PROGRAM Stn054_29_EmptyPuckStorageMergeGrn
VAR
	{attribute 'TcLinkToOSO' := '	
			.iBufferFull :=  <0,1,3>TIIB[N56S00 (AL1332)]^N56S05 (AL2341)^TxPDO^input byte 2'}
	fbConvMerge: FB_ConvMerge_RemoteOutput;
	
	{attribute 'TcLinkToOSO' := '
			<0,1,3>TIIB[N56S00 (AL1332)]^N56S05 (AL2341)^TxPDO^input byte 2'}
	iBufferFull AT %I*: BOOL;

END_VAR

//  This code instantiates a component that is implimented as a common function block
//    Note that I/O is linked directly to I/O variables inside the named instance
// This merge is NOT linked to any work cell

gStn054_29_EmptyPuckStorageMergeGrn.MainHeartbeatOK := TRUE; // because this PLC is Main
gStn054_29_EmptyPuckStorageMergeGrn.MainConvRunning := gConsumed_SafetyInterfaceConv.MtrRunning.Enc058Mtr05;
gStn054_29_EmptyPuckStorageMergeGrn.MainInAuto := gStn054.CycleAuto;

gStn054_29_EmptyPuckStorageMergeGrn.SpurHeartbeatOK := TRUE;  //because this PLC is Main
gStn054_29_EmptyPuckStorageMergeGrn.SpurConvRunning := gConsumed_SafetyInterfaceConv.MtrRunning.Enc058Mtr05 AND  gConsumed_SafetyInterfaceConv.MtrRunning.Enc058Mtr03;
gStn054_29_EmptyPuckStorageMergeGrn.SpurInAuto := gStn054.CycleAuto; 

fbConvMerge(
	pStn := ADR(gStn054),
	pCmp := ADR(gStn054_29_EmptyPuckStorageMergeGrn),
	pStateTraceBuffer := ADR(gStn054_StateTraceBuffer),
	pStateTraceFifo := ADR(gStn054_StateTraceFifo),
	pStats := ADR(gStn054_02_Stats),
	pMain := ADR(gStn054_27_EmptyPuckStorageMainMergePrestopGrn),
	pSpur := ADR(gStn054_28_EmptyPuckStorageSpurMergePrestopGrn)		
);

END_PROGRAM

(* stored: Version 1.1.0.1, ProductVersion 3.1.4024.6
   POU Stn054_29_EmptyPuckStorageMergeGrn: Id {71de74b4-c432-4519-86fc-29544f2c1950}, SpecialFunc None *)
